{attribute 'qualified_only'}
VAR_GLOBAL PERSISTENT
	totalRunHours : LREAL := 0;
END_VAR

(* stored: Version 1.1.0.1, ProductVersion 3.1.4024.12
   GVL GVL_OperationCounter: Id {8cc793b9-a930-4453-96af-f928e3127afd} *)
